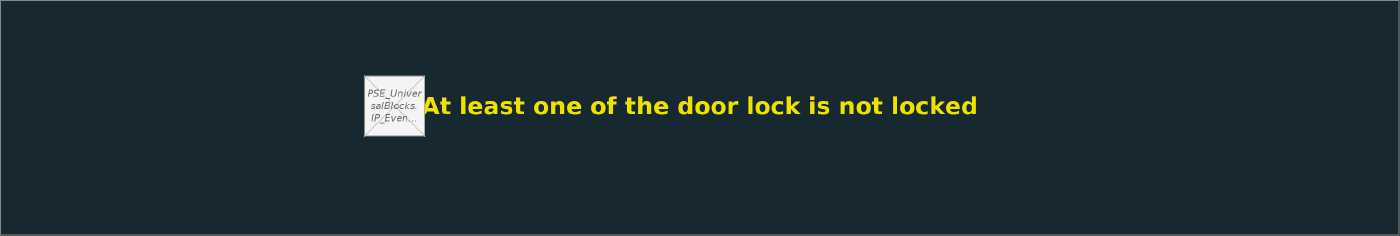
VISUALIZATION InitializingDoorLockOpen  // 1480x250
    Label (0,92 1480x40), "At least one of the door lock is not locked"
    Image (385,80 64x64), image: PSE_UniversalBlocks.IP_EventSeverity.error
END_VISUALIZATION

(* stored: Version 1.1.0.1, ProductVersion 3.1.4024.9
   Visu InitializingDoorLockOpen: Id {5fac8ee8-eebf-4c01-84b9-c2ba9ec6621f} *)
